// TwinCAT 3 PLC project basic_motor_control
// ProgramVersion: 3.1.4023.0
// libraries:
//   Tc2_Standard, * (Beckhoff Automation GmbH)
//   Tc2_System, * (Beckhoff Automation GmbH)
//   Tc3_Module, * (Beckhoff Automation GmbH)
// project tree:
//   GVLs/ GVL.TcGVL
//   / PlcTask.TcTTO
//   POUs/ MAIN.TcPOU
// real-time tasks:
//   TASK PlcTask: cycle T#10ms, priority 20, ADS port 350

CONFIGURATION basic_motor_control
    RESOURCE PLC ON TwinCAT3
        TASK PlcTask(INTERVAL := T#10ms, PRIORITY := 20);
        PROGRAM MAIN WITH PlcTask : MAIN;
    END_RESOURCE
END_CONFIGURATION

// ---- GVLs/GVL.TcGVL
{attribute 'qualified_only'}
VAR_GLOBAL
	



END_VAR

// ---- POUs/MAIN.TcPOU
PROGRAM MAIN
VAR
	MyBoolean : BOOL;
	MyBoolean_2: BOOL;
	
	MyInt : INT;
	MyInt_2 : INT;
	
END_VAR



MyBoolean := TRUE;
MyInt:=3;

END_PROGRAM
